FUNCTION_BLOCK FB_VisionOrientation EXTENDS FB_PackML_BaseModule
VAR
	SpinAxis			: FB_Component_BasicAxis;
	Camera				: FB_PlcCameraBase;
	TON_Delay			: TON;
	_SpinAxisPositionModulo	: LREAL;
	ImageCaptureAngle	: LREAL := 130;
	SpinVelocity		: LREAL := 500;
END_VAR

//! @summary This method contains code which will execute when this PackML module is in the <b>Aborting</b> state
METHOD PROTECTED Aborting
VAR
	i				: UDINT;
	SubModulesReady : BOOL := TRUE;
END_VAR
CASE DescendantSequenceState OF
	0:
		NoStateTasksToComplete := FALSE;
		DescendantSequenceState := DescendantSequenceState + 10;

	10:
		IF SpinAxis.Disable() THEN
			StateTasksComplete 		:= TRUE;
			DescendantSequenceState := DescendantSequenceState + 10;
		END_IF

	20:
		StateTasksComplete := TRUE;
END_CASE

SUPER^.Aborting();
END_METHOD

//! @summary This method contains code which will execute when this PackML module is in the <b>Clearing</b> state
METHOD PROTECTED Clearing
VAR
	i				: UDINT;
	SubModulesReady : BOOL := TRUE;
END_VAR

VAR_INST

END_VAR

(*! <description> <b>Note:</b> The <i>Clear</i> command can also be thought of as a <i>fault reset</i> depite the ambiguity in the naming of the <i>Reset</i> state. 
<table> 
	<tr>
		<th> Previous State </th>
		<th> Transition In </th>
		<th> Transition Out </th>
		<th> Next State  </th> 
	</tr>
	<tr>
		<td> Aborted </td>
		<td> Clear Command </td> 
		<td> State Complete </td>
		<td> Stopped </td> 
	</tr>
</table>
This method is called as required by <c>StateControl()</c>
</description> 

*)
// CASE _CurrentMode OF
// 	E_PMLUnitMode.ePMLUnitMode_Production:
		CASE DescendantSequenceState OF
			0: //Init
				NoStateTasksToComplete := FALSE;

				//Reset Axes and  CA Group
				SpinAxis.Reset();
				DescendantSequenceState := DescendantSequenceState + 10;

			10: // Done	
				StateTasksComplete := TRUE;
		END_CASE

// END_CASE

SUPER^.Clearing();
END_METHOD

METHOD CyclicLogic
VAR_INPUT
END_VAR
SUPER^.CyclicLogic();

TON_Delay();
END_METHOD

//! @summary This method contains code which will execute when this PackML module is in the <b>Execute</b> state
METHOD PROTECTED Execute
VAR
	i : UDINT;
END_VAR
CASE DescendantSequenceState OF
	0:	// Start Spinning
		SpinAxis.MoveVelocity(SpinVelocity, TRUE);
		TON_Delay.IN				:= TRUE;
		DescendantSequenceState		:= DescendantSequenceState + 10;

	10:	// Trigger Images bad way
		IF TON_Delay.Q THEN
			IF SpinAxis.SetPositionModulo > ImageCaptureAngle AND _SpinAxisPositionModulo < ImageCaptureAngle THEN

				// Trigger Image
				Camera.TriggerImage	:= TRUE;

				TON_Delay(IN 		:= FALSE);
				TON_Delay.IN		:= TRUE;
			END_IF
		ELSE
			Camera.TriggerImage		:= FALSE;
		END_IF

	20:	// Trigger Images good way
		IF TON_Delay.Q THEN
			IF SpinAxis.SetPositionModulo > ImageCaptureAngle AND _SpinAxisPositionModulo < ImageCaptureAngle THEN

				// Trigger Image
				Camera.TriggerImage	:= TRUE;

				// for xfc
				// add slots to camera process image
				// xfc fb will output time
				// convert that to ulint with fb called "extenddctime" or similar
				// sent that dc time off to camera

				// xfc fb is non-modulo, so need to modulo 
				// modturns is a funcation that calculates the number of turns, to un-modulo a target position (in tc2_math)
				// tc2_math also has mod_abs that takes absolute position and modulo factor and tells you where in modulo position you are
				

				TON_Delay(IN 		:= FALSE);
				TON_Delay.IN		:= TRUE;
			END_IF
		ELSE
			Camera.TriggerImage		:= FALSE;
		END_IF


END_CASE

_SpinAxisPositionModulo	:= SpinAxis.SetPositionModulo;
END_METHOD

(* Basic module initialization logic*)
METHOD PROTECTED Initialize : BOOL
Initialize := FALSE;
CASE DescendantSequenceState OF
	0:
		RegisterComponent(Component := SpinAxis);
		RegisterComponent(Component := Camera);
		DescendantSequenceState := DescendantSequenceState + 10;

	10:
		IF SUPER^.Initialize() THEN
			DescendantSequenceState := DescendantSequenceState + 10;
		END_IF

	20:
		Initialize := TRUE;
END_CASE
END_METHOD

METHOD PROTECTED Resetting
VAR_INST
	i			 : UDINT;
END_VAR
CASE DescendantSequenceState OF
	0: //Init
		NoStateTasksToComplete := FALSE;
		DescendantSequenceState := DescendantSequenceState + 10;

	10: //Reset Everything
		IF SpinAxis.Enable() AND Camera.Reset() THEN
			DescendantSequenceState := DescendantSequenceState + 10;
		END_IF

	20: //Clearing complete
		StateTasksComplete := TRUE;

END_CASE

SUPER^.Resetting();
END_METHOD

METHOD PROTECTED Starting
CASE DescendantSequenceState OF
	0:
		NoStateTasksToComplete	:= FALSE;
		DescendantSequenceState := 10;

	10: //Set Axis Parameters
		SpinAxis.Velocity		:= 180;
		SpinAxis.Acceleration	:= 360;
		SpinAxis.Deceleration	:= 360;
		SpinAxis.Jerk			:= 1000;
		TON_Delay.PT			:= T#1S;
		DescendantSequenceState := DescendantSequenceState + 10;

	20: // Start Running Vision
		Camera.RunVision		:= TRUE;
		DescendantSequenceState := DescendantSequenceState + 10;

	30: // check that vision is running
		IF Camera.CameraState = TCVN_CS_ACQUIRING THEN
			DescendantSequenceState := DescendantSequenceState + 10;
		END_IF

	40: //Cleanup mover queues
		StateTasksComplete 		:= TRUE;

END_CASE

SUPER^.Starting();
END_METHOD

(* This method contains code which will execute when this PackML module is in the Stopping state*)
METHOD PROTECTED Stopping
CASE DescendantSequenceState OF
	0:
		NoStateTasksToComplete	:= FALSE;
		DescendantSequenceState := 10;

	10: //Set Axis Parameters
		SpinAxis.Stop();
		TON_Delay.IN		:= FALSE;
		Camera.TriggerImage	:= FALSE;
		DescendantSequenceState := DescendantSequenceState + 10;

	20: //Cleanup mover queues
		StateTasksComplete 		:= TRUE;

END_CASE

SUPER^.Stopping();
END_METHOD

END_FUNCTION_BLOCK

(* stored: Version 1.1.0.1
   POU FB_VisionOrientation: Id {448371c6-13eb-43c4-a0ce-ebb192d17413}, SpecialFunc None
   Folder Acting States: Id {e14cf1b1-45ff-4fb4-81b9-1f52a5d32669}
   Folder Waiting States: Id {ab86d3ba-50da-471d-864b-21041ca20d53}
   Method Aborting: Id {08b82fb7-4aad-43b5-9009-69587d93ae28}
   Method Clearing: Id {00b4c057-1c77-497e-ad7c-49ae2f8309bf}
   Method CyclicLogic: Id {f349efda-102a-4c03-85f1-b156c57de820}
   Method Execute: Id {4a8447c7-4bba-456b-ae99-02b9655bd430}
   Method Initialize: Id {735d1fea-bfd6-4ba8-b1c5-4688da7cba47}
   Method Resetting: Id {c9015cb7-7c60-4a02-a992-009fb7a3167f}
   Method Starting: Id {0102240e-1ac7-403e-9ddc-852ca008333e}
   Method Stopping: Id {f363e253-5d73-436d-a63d-0518e246a925} *)
